// TIA Portal V15.1 export
// export: Created 2026-01-09T13:45:12.0760408Z, ExportSetting WithDefaults, WithReadOnly, DisplayName Totally Integrated Automation Portal, DisplayVersion V15.1 Update 8, DisplayName TIA Portal Openness, DisplayVersion V15.1 Update 8, DisplayName STEP 7 Professional, DisplayVersion V15.1 Update 8, DisplayName WinCC Advanced, DisplayVersion V15.1 Update 8
FUNCTION_BLOCK "2.MANUAL_CONTROL"   // FB2, LAD
TITLE = MODE=0 thì nhấn dạng Toggle, MODE=1 thì nhấn như một nút nhấn thông thường, nếu RS=1 thì ngõ ra sẽ bị Reset
{ S7_Optimized_Access := 'TRUE' }
VERSION : 0.1
// Chức năng của FB: xác định phương thức tác động khi nhấn nút NN1, NN2, NN3 theo 2 cách
// Cách 1: MODE = 0, thực hiện như một Toggle, mỗi lần nhấn sẽ đổi trạng thái OUT, từ OFF sang ON và ngược lại.
// NN là nút nhấn trên HMI/SCADA
// OUT là ngõ ra cần được SET hoặc RESET
// ST chính là OUT (nó như là phản hồi để biết OUT đang được SET hay RESET
// RS là tín hiệu để reset ngõ ra
// Nó dùng M là một biến Static để lưu số lần nhấn nút (ban đầu nếu chưa có ngõ ra OUT, thì M là 0, nhưng khi đã có OUT thì M  là 1), từ đây nếu NN nhấn mà chưa có OUT thì OUT11 sẽ được SET, còn nếu NN được nhấn mà có OUT11 thì sẽ Reset OUT11 đi)
// Cách 2: MODE=1, nó thực hiện như một nút nhấn mình thường dạng Momentory, nghĩa là Nhấn thì đầu ra sẽ có, còn nhả ra thì mất OUT.
// stored: AutoNumber false, CodeModifiedDate 2025-08-27T17:14:33.2091456Z, CompileDate 2025-08-30T17:40:32.4655936Z, CreationDate 2024-10-12T12:36:08.0193576Z, DownloadWithoutReinit false, HandleErrorsWithinBlock false, InterfaceModifiedDate 2025-08-27T17:14:33.2091456Z, IsConsistent true, IsIECCheckEnabled false, IsKnowHowProtected false, IsRetainMemResEnabled false, IsWriteProtected false, LibraryConformanceStatus The object is library-conformant., MemoryReserve 100, ModifiedDate 2025-10-23T13:27:09.8211701Z, ParameterModified 2024-10-13T14:59:19.5830719Z, PLCSimAdvancedSupport false, SetENOAutomatically False, StructureModified 2025-08-27T17:14:33.2091456Z, UDAEnableTagReadback false
   VAR_INPUT
      MODE : Bool;
      NN1 : Bool;
      NN2 : Bool;
      NN3 : Bool;
      ST1 : Bool;
      ST2 : Bool;
      ST3 : Bool;
      RS1 : Bool;
      RS2 : Bool;
      RS3 : Bool;
   END_VAR
   VAR_OUTPUT
      OUT1 : Bool;
      OUT2 : Bool;
      OUT3 : Bool;
   END_VAR
   VAR
      OUT11 : Bool;
      OUT12 : Bool;
      OUT21 : Bool;
      OUT22 : Bool;
      OUT31 : Bool;
      OUT32 : Bool;
      M1 : Int;
      M2 : Int;
      M3 : Int;
      M4 : Bool;
      M5 : Bool;
      M6 : Bool;
   END_VAR
   VAR_TEMP
      T1 : Bool;
      T2 : Bool;
      T3 : Bool;
      T4 : Bool;
      T5 : Bool;
      T6 : Bool;
   END_VAR
   VAR_TEMP   // added for the SCL form of the ladder/FBD networks
      _w1 : Bool;
   END_VAR
BEGIN

REGION Network 1
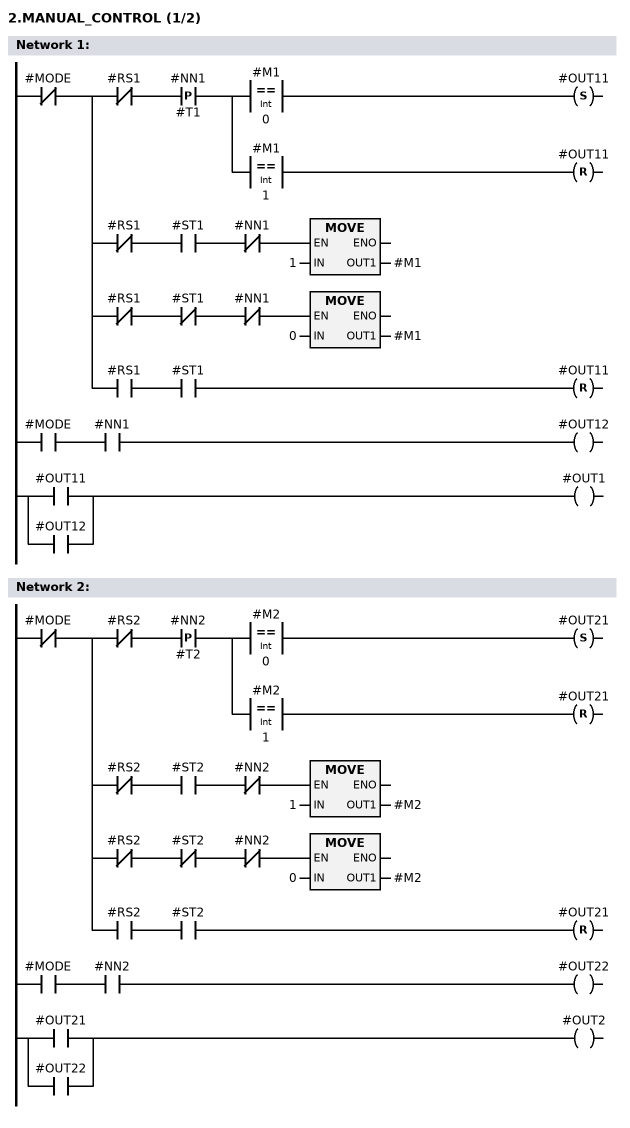
   RUNG wire#powerrail
      I_Contact( #MODE )
      wire#w1
      I_Contact( #RS1 )
      P_Contact(operand := #NN1, bit := #T1)
      wire#w2
      { S7_Templates := "SrcType := Int" } EQ_Contact(in1 := #M1, in2 := 0)
      S_Coil( #OUT11 )
   END_RUNG
   RUNG wire#w2
      { S7_Templates := "SrcType := Int" } EQ_Contact(in1 := #M1, in2 := 1)
      R_Coil( #OUT11 )
   END_RUNG
   RUNG wire#w1
      I_Contact( #RS1 )
      Contact( #ST1 )
      I_Contact( #NN1 )
      Move(in := 1, out1 => #M1)
   END_RUNG
   RUNG wire#w1
      I_Contact( #RS1 )
      I_Contact( #ST1 )
      I_Contact( #NN1 )
      Move(in := 0, out1 => #M1)
   END_RUNG
   RUNG wire#w1
      Contact( #RS1 )
      Contact( #ST1 )
      R_Coil( #OUT11 )
   END_RUNG
   RUNG wire#powerrail
      Contact( #MODE )
      Contact( #NN1 )
      Coil( #OUT12 )
   END_RUNG
   RUNG wire#powerrail
      Contact( #OUT11 )
      wire#w3
      Coil( #OUT1 )
   END_RUNG
   RUNG wire#powerrail
      Contact( #OUT12 )
   END_RUNG wire#w3
   // the same network as SCL:
   #_w1 := NOT #MODE AND NOT #RS1 AND #NN1 AND NOT #T1;   // rising edge of #NN1
   #T1 := #NN1;
   IF #_w1 AND (#M1 = 0) THEN #OUT11 := TRUE; END_IF;
   IF #_w1 AND (#M1 = 1) THEN #OUT11 := FALSE; END_IF;
   IF NOT #MODE AND NOT #RS1 AND #ST1 AND NOT #NN1 THEN #M1 := 1; END_IF;
   IF NOT #MODE AND NOT #RS1 AND NOT #ST1 AND NOT #NN1 THEN #M1 := 0; END_IF;
   IF NOT #MODE AND #RS1 AND #ST1 THEN #OUT11 := FALSE; END_IF;
   #OUT12 := #MODE AND #NN1;
   #OUT1 := #OUT11 OR #OUT12;
END_REGION

REGION Network 2
   RUNG wire#powerrail
      I_Contact( #MODE )
      wire#w1
      I_Contact( #RS2 )
      P_Contact(operand := #NN2, bit := #T2)
      wire#w2
      { S7_Templates := "SrcType := Int" } EQ_Contact(in1 := #M2, in2 := 0)
      S_Coil( #OUT21 )
   END_RUNG
   RUNG wire#w2
      { S7_Templates := "SrcType := Int" } EQ_Contact(in1 := #M2, in2 := 1)
      R_Coil( #OUT21 )
   END_RUNG
   RUNG wire#w1
      I_Contact( #RS2 )
      Contact( #ST2 )
      I_Contact( #NN2 )
      Move(in := 1, out1 => #M2)
   END_RUNG
   RUNG wire#w1
      I_Contact( #RS2 )
      I_Contact( #ST2 )
      I_Contact( #NN2 )
      Move(in := 0, out1 => #M2)
   END_RUNG
   RUNG wire#w1
      Contact( #RS2 )
      Contact( #ST2 )
      R_Coil( #OUT21 )
   END_RUNG
   RUNG wire#powerrail
      Contact( #MODE )
      Contact( #NN2 )
      Coil( #OUT22 )
   END_RUNG
   RUNG wire#powerrail
      Contact( #OUT21 )
      wire#w3
      Coil( #OUT2 )
   END_RUNG
   RUNG wire#powerrail
      Contact( #OUT22 )
   END_RUNG wire#w3
   // the same network as SCL:
   #_w1 := NOT #MODE AND NOT #RS2 AND #NN2 AND NOT #T2;   // rising edge of #NN2
   #T2 := #NN2;
   IF #_w1 AND (#M2 = 0) THEN #OUT21 := TRUE; END_IF;
   IF #_w1 AND (#M2 = 1) THEN #OUT21 := FALSE; END_IF;
   IF NOT #MODE AND NOT #RS2 AND #ST2 AND NOT #NN2 THEN #M2 := 1; END_IF;
   IF NOT #MODE AND NOT #RS2 AND NOT #ST2 AND NOT #NN2 THEN #M2 := 0; END_IF;
   IF NOT #MODE AND #RS2 AND #ST2 THEN #OUT21 := FALSE; END_IF;
   #OUT22 := #MODE AND #NN2;
   #OUT2 := #OUT21 OR #OUT22;
END_REGION

REGION Network 3
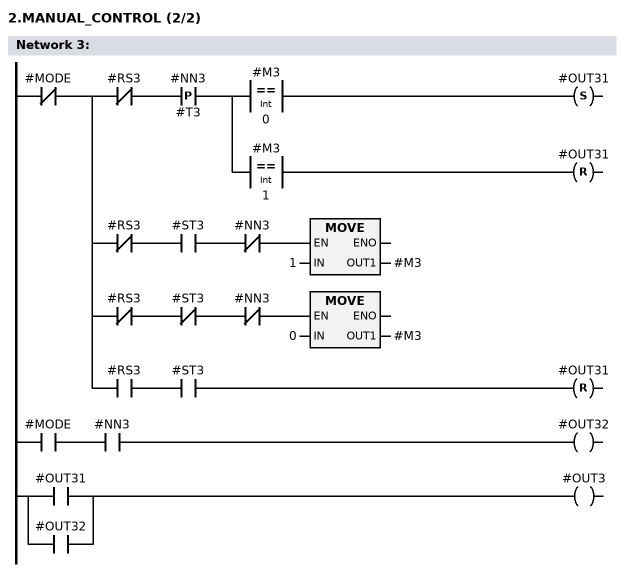
   RUNG wire#powerrail
      I_Contact( #MODE )
      wire#w1
      I_Contact( #RS3 )
      P_Contact(operand := #NN3, bit := #T3)
      wire#w2
      { S7_Templates := "SrcType := Int" } EQ_Contact(in1 := #M3, in2 := 0)
      S_Coil( #OUT31 )
   END_RUNG
   RUNG wire#w2
      { S7_Templates := "SrcType := Int" } EQ_Contact(in1 := #M3, in2 := 1)
      R_Coil( #OUT31 )
   END_RUNG
   RUNG wire#w1
      I_Contact( #RS3 )
      Contact( #ST3 )
      I_Contact( #NN3 )
      Move(in := 1, out1 => #M3)
   END_RUNG
   RUNG wire#w1
      I_Contact( #RS3 )
      I_Contact( #ST3 )
      I_Contact( #NN3 )
      Move(in := 0, out1 => #M3)
   END_RUNG
   RUNG wire#w1
      Contact( #RS3 )
      Contact( #ST3 )
      R_Coil( #OUT31 )
   END_RUNG
   RUNG wire#powerrail
      Contact( #MODE )
      Contact( #NN3 )
      Coil( #OUT32 )
   END_RUNG
   RUNG wire#powerrail
      Contact( #OUT31 )
      wire#w3
      Coil( #OUT3 )
   END_RUNG
   RUNG wire#powerrail
      Contact( #OUT32 )
   END_RUNG wire#w3
   // the same network as SCL:
   #_w1 := NOT #MODE AND NOT #RS3 AND #NN3 AND NOT #T3;   // rising edge of #NN3
   #T3 := #NN3;
   IF #_w1 AND (#M3 = 0) THEN #OUT31 := TRUE; END_IF;
   IF #_w1 AND (#M3 = 1) THEN #OUT31 := FALSE; END_IF;
   IF NOT #MODE AND NOT #RS3 AND #ST3 AND NOT #NN3 THEN #M3 := 1; END_IF;
   IF NOT #MODE AND NOT #RS3 AND NOT #ST3 AND NOT #NN3 THEN #M3 := 0; END_IF;
   IF NOT #MODE AND #RS3 AND #ST3 THEN #OUT31 := FALSE; END_IF;
   #OUT32 := #MODE AND #NN3;
   #OUT3 := #OUT31 OR #OUT32;
END_REGION
END_FUNCTION_BLOCK
